{attribute 'qualified_only'}
TYPE ErrorCode :
(
	SUCCESS := 0,
	
	// Preparation Error 
	PREPARATION_DONE := 1000,
	PREPARATION_WATER_HIGH_TEMP,
	PREPARATION_FLAME,
	PREPARATION_PUMP_NOT_CONNECTED,
	
	// Ignition Error
	IGNITION_DONE := 2000,
	IGNITION_FLAME,
	
	// Burning Error
	BURNING_DONE := 3000,
	BURNING_EMERGENCY_TEMPERATURE,
	
	// Stop Error
	STOP_ERROR	:= 4000
) UINT;
END_TYPE

(* stored: Version 1.1.0.1, ProductVersion 3.1.4022.18
   DUT ErrorCode: Id {ef136dff-3693-4972-84b7-ce647f7dd58d} *)
